(* PLC project PLCopen TC2 library, Higen Motion Controller 0.0 *)
(* stored: creationDateTime 2011-12-10T00:00:00, modificationDateTime 2011-12-10T00:00:00 *)

TYPE AXIS_REF : INT := -1;
END_TYPE

TYPE MC_BUFFER_MODE : (mcAborting, mcBuffered, mcBlendingLow, mcBlendingPrevious, mcBlendingNext, mcBlendingHigh) := mcAborting;
END_TYPE

TYPE MC_HOMING_PROCEDURES : (mcHomeDirect, mcHomeLimitSwitchPositive, mcHomeLimitSwitchNegative, mcHomeAbsoluteSwitchPositive, mcHomeAbsoluteSwitchNegative, mcHomeReferencePulsePositive, mcHomeReferencePulseNegative, mcHomeAbsolute) := mcHomeDirect;
END_TYPE

TYPE MC_DIRECTION : (mcAbsolutePosition, mcPositiveDirection, mcShortestWay, mcNegativeDirection, mcCurrentDirection) := mcAbsolutePosition;
END_TYPE

TYPE MC_TP_REF : INT := -1;
END_TYPE

TYPE MC_TV_REF : INT := -1;
END_TYPE

TYPE MC_TA_REF : INT := -1;
END_TYPE

TYPE MC_EXECUTION_MODE : (mcImmediately, mcQueued) := mcImmediately;
END_TYPE

TYPE MC_SOURCE : (mcActualValue, mcSetValue) := mcActualValue;
END_TYPE

TYPE MC_CAMSWITCH_REF : INT := -1;
END_TYPE

TYPE MC_OUTPUT_REF : INT := -1;
END_TYPE

TYPE MC_TRACK_REF : INT := -1;
END_TYPE

TYPE MC_TRIGGER_REF : INT := -1;
END_TYPE

TYPE MC_CAM_REF : INT := -1;
END_TYPE

TYPE MC_CAM_ID : INT := -1;
END_TYPE

TYPE MC_START_MODE : INT := -1;
END_TYPE

TYPE MC_SYNC_MODE : INT := -1;
END_TYPE

TYPE MC_COMBINE_MODE : (mcAddAxes, mcSubAxes) := mcAddAxes;
END_TYPE

TYPE MC_REAL_ARRAY : ARRAY[1..6] OF LREAL;
END_TYPE

TYPE MC_INT_ARRAY : ARRAY[1..6] OF INT;
END_TYPE

(* This fonction blocks returns the axis torque limits *)
FUNCTION_BLOCK MC_GetTorqueLimit
  VAR_IN_OUT
    Axis : AXIS_REF;
  END_VAR
  VAR_INPUT
    Execute : BOOL;
  END_VAR
  VAR_OUTPUT
    Done : BOOL;
    Busy : BOOL;
    Error : BOOL;
    ErrorID : WORD;
  END_VAR
  VAR_OUTPUT
    TorqueLimitPos : UINT;
    TorqueLimitNeg : UINT;
  END_VAR
  VAR
    Execute0 : BOOL;
    Done0 : BOOL;
  END_VAR

    {{
    extern void __mcl_cmd_MC_GetTorqueLimit(MC_GETTORQUELIMIT*);
    __mcl_cmd_MC_GetTorqueLimit(data__);
    }}
    Execute0 := Execute;
    Done0 := Done;
END_FUNCTION_BLOCK

(* This fonction blocks defines the axis torque limits *)
FUNCTION_BLOCK MC_SetTorqueLimit
  VAR_IN_OUT
    Axis : AXIS_REF;
  END_VAR
  VAR_INPUT
    Execute : BOOL;
  END_VAR
  VAR_OUTPUT
    Done : BOOL;
    Busy : BOOL;
    Error : BOOL;
    ErrorID : WORD;
  END_VAR
  VAR_INPUT
    TorqueLimitPos : UINT;
    TorqueLimitNeg : UINT;
  END_VAR
  VAR
    Execute0 : BOOL;
    Done0 : BOOL;
  END_VAR

    {{
    extern void __mcl_cmd_MC_SetTorqueLimit(MC_SETTORQUELIMIT*);
    __mcl_cmd_MC_SetTorqueLimit(data__);
    }}
    Execute0 := Execute;
    Done0 := Done;
END_FUNCTION_BLOCK

(* This Function Block controls the power stage (On or Off). *)
FUNCTION_BLOCK MC_Power
  VAR_IN_OUT
    Axis : AXIS_REF;
  END_VAR
  VAR_INPUT
    Enable : BOOL;
    EnablePositive : BOOL;
    EnableNegative : BOOL;
  END_VAR
  VAR_OUTPUT
    Status : BOOL;
    Valid : BOOL;
    Error : BOOL;
    ErrorID : WORD;
  END_VAR

    {{
    extern void __mcl_cmd_MC_Power(MC_POWER*);
    __mcl_cmd_MC_Power(data__);
    }}
END_FUNCTION_BLOCK

(* This Function Block commands the axis to perform the «search home» sequence. The details of this sequence are manufacturer dependent and can be set by the axis’ parameters. The ‘Position’ input is used to set the absolute position when reference signal is detected. This Function Block completes at ‘Standstill’ if it was started in ‘Standstill’. *)
FUNCTION_BLOCK MC_Home
  VAR_IN_OUT
    Axis : AXIS_REF;
  END_VAR
  VAR_INPUT
    Execute : BOOL;
    Position : LREAL;
    HomingMode : MC_HOMING_PROCEDURES;
    BufferMode : MC_BUFFER_MODE;
  END_VAR
  VAR_OUTPUT
    Done : BOOL;
    Busy : BOOL;
    Active : BOOL;
    CommandAborted : BOOL;
    Error : BOOL;
    ErrorID : WORD;
  END_VAR
  VAR
    Execute0 : BOOL;
    Done0 : BOOL;
    Active0 : BOOL;
  END_VAR

    {{
    extern void __mcl_cmd_MC_Home(MC_HOME*);
    __mcl_cmd_MC_Home(data__);
    }}
    Execute0 := Execute;
    Done0 := Done;
END_FUNCTION_BLOCK

(* This Function Block commands a controlled motion stop and transfers the axis to the state ‘Stopping’. It aborts any ongoing Function Block execution. While the axis is in state ‘Stopping’, no other FB can perform any motion on the same axis. After the axis has reached ‘Velocity’ zero, the ‘Done’ output is set to TRUE immediately. The axis remains in the state ‘Stopping’ as long as ‘Execute’ is still TRUE or ‘Velocity’ zero is not yet reached. As soon as ‘Done’ is SET and ‘Execute’ is FALSE the axis goes to state ‘Standstill’. *)
FUNCTION_BLOCK MC_Stop
  VAR_IN_OUT
    Axis : AXIS_REF;
  END_VAR
  VAR_INPUT
    Execute : BOOL;
    Deceleration : LREAL;
    Jerk : LREAL;
  END_VAR
  VAR_OUTPUT
    Done : BOOL;
    Busy : BOOL;
    CommandAborted : BOOL;
    Error : BOOL;
    ErrorID : WORD;
  END_VAR
  VAR
    Execute0 : BOOL;
    Done0 : BOOL;
    Active0 : BOOL;
  END_VAR

    {{
    extern void __mcl_cmd_MC_Stop(MC_STOP*);
    __mcl_cmd_MC_Stop(data__);
    }}
    Execute0 := Execute;
    Done0 := Done;
END_FUNCTION_BLOCK

(* This Function Block commands a controlled motion stop. The axis is moved to the state ‘DiscreteMotion’, until the velocity is zero. With the ‘Done’ output set, the state is transferred to ‘Standstill’. *)
FUNCTION_BLOCK MC_Halt
  VAR_IN_OUT
    Axis : AXIS_REF;
  END_VAR
  VAR_INPUT
    Execute : BOOL;
    Deceleration : LREAL;
    Jerk : LREAL;
    BufferMode : MC_BUFFER_MODE;
  END_VAR
  VAR_OUTPUT
    Done : BOOL;
    Busy : BOOL;
    Active : BOOL;
    CommandAborted : BOOL;
    Error : BOOL;
    ErrorID : WORD;
  END_VAR
  VAR
    Execute0 : BOOL;
    Done0 : BOOL;
    Active0 : BOOL;
  END_VAR

    {{
    extern void __mcl_cmd_MC_Halt(MC_HALT*);
    __mcl_cmd_MC_Halt(data__);
    }}
    Execute0 := Execute;
    Done0 := Done;
END_FUNCTION_BLOCK

(* This Function Block commands a controlled motion to a specified absolute position. *)
FUNCTION_BLOCK MC_MoveAbsolute
  VAR_IN_OUT
    Axis : AXIS_REF;
  END_VAR
  VAR_INPUT
    Execute : BOOL;
    ContinuousUpdate : BOOL;
    Position : LREAL;
    Velocity : LREAL;
    Acceleration : LREAL;
    Deceleration : LREAL;
    Jerk : LREAL;
    Direction : MC_DIRECTION;
    BufferMode : MC_BUFFER_MODE;
  END_VAR
  VAR_OUTPUT
    Done : BOOL;
    Busy : BOOL;
    Active : BOOL;
    CommandAborted : BOOL;
    Error : BOOL;
    ErrorID : WORD;
  END_VAR
  VAR
    Execute0 : BOOL;
    Done0 : BOOL;
    Active0 : BOOL;
  END_VAR

    {{
    extern void __mcl_cmd_MC_MoveAbsolute(MC_MOVEABSOLUTE*);
    __mcl_cmd_MC_MoveAbsolute(data__);
    }}
    Execute0 := Execute;
    Done0 := Done;
END_FUNCTION_BLOCK

(* This Function Block commands a controlled motion of a specified distance relative to the set position at the time of the execution. *)
FUNCTION_BLOCK MC_MoveRelative
  VAR_IN_OUT
    Axis : AXIS_REF;
  END_VAR
  VAR_INPUT
    Execute : BOOL;
    ContinuousUpdate : BOOL;
    Distance : LREAL;
    Velocity : LREAL;
    Acceleration : LREAL;
    Deceleration : LREAL;
    Jerk : LREAL;
    BufferMode : MC_BUFFER_MODE;
  END_VAR
  VAR_OUTPUT
    Done : BOOL;
    Busy : BOOL;
    Active : BOOL;
    CommandAborted : BOOL;
    Error : BOOL;
    ErrorID : WORD;
  END_VAR
  VAR
    Execute0 : BOOL;
    Done0 : BOOL;
    Active0 : BOOL;
  END_VAR

    {{
    extern void __mcl_cmd_MC_MoveRelative(MC_MOVERELATIVE*);
    __mcl_cmd_MC_MoveRelative(data__);
    }}
    Execute0 := Execute;
    Done0 := Done;
END_FUNCTION_BLOCK

(* This Function Block commands a controlled motion of a specified relative distance additional to the most recent commanded position in the axis state ‘DiscreteMotion’. The most recent commanded position may be the result of a previous MC_MoveAdditive motion which was aborted. If the FB is activated in the axis state ‘ContinuousMotion’, the specified relative distance is added to the set position at the time of the execution. *)
FUNCTION_BLOCK MC_MoveAdditive
  VAR_IN_OUT
    Axis : AXIS_REF;
  END_VAR
  VAR_INPUT
    Execute : BOOL;
    ContinuousUpdate : BOOL;
    Distance : LREAL;
    Velocity : LREAL;
    Acceleration : LREAL;
    Deceleration : LREAL;
    Jerk : LREAL;
    BufferMode : MC_BUFFER_MODE;
  END_VAR
  VAR_OUTPUT
    Done : BOOL;
    Busy : BOOL;
    Active : BOOL;
    CommandAborted : BOOL;
    Error : BOOL;
    ErrorID : WORD;
  END_VAR
  VAR
    Execute0 : BOOL;
    Done0 : BOOL;
    Active0 : BOOL;
  END_VAR

    {{
    extern void __mcl_cmd_MC_MoveAdditive(MC_MOVEADDITIVE*);
    __mcl_cmd_MC_MoveAdditive(data__);
    }}
    Execute0 := Execute;
    Done0 := Done;
END_FUNCTION_BLOCK

(* This Function Block commands a controlled motion of a specified relative distance additional to an existing motion. The existing Motion is not interrupted, but is superimposed by the additional motion. *)
FUNCTION_BLOCK MC_MoveSuperimposed
  VAR_IN_OUT
    Axis : AXIS_REF;
  END_VAR
  VAR_INPUT
    Execute : BOOL;
    ContinuousUpdate : BOOL;
    Distance : LREAL;
    VelocityDiff : LREAL;
    Acceleration : LREAL;
    Deceleration : LREAL;
    Jerk : LREAL;
  END_VAR
  VAR_OUTPUT
    Done : BOOL;
    Busy : BOOL;
    CommandAborted : BOOL;
    Error : BOOL;
    ErrorID : WORD;
    CoveredDistance : LREAL;
  END_VAR
  VAR
    Execute0 : BOOL;
    Done0 : BOOL;
    Active0 : BOOL;
  END_VAR

    {{
    extern void __mcl_cmd_MC_MoveSuperimposed(MC_MOVESUPERIMPOSED*);
    __mcl_cmd_MC_MoveSuperimposed(data__);
    }}
    Execute0 := Execute;
    Done0 := Done;
END_FUNCTION_BLOCK

(* This Function Block commands a halt to all superimposed motions of the axis. The underlying motion is not interrupted. *)
FUNCTION_BLOCK MC_HaltSuperimposed
  VAR_IN_OUT
    Axis : AXIS_REF;
  END_VAR
  VAR_INPUT
    Execute : BOOL;
    Deceleration : LREAL;
    Jerk : LREAL;
  END_VAR
  VAR_OUTPUT
    Done : BOOL;
    Busy : BOOL;
    CommandAborted : BOOL;
    Error : BOOL;
    ErrorID : WORD;
  END_VAR
  VAR
    Execute0 : BOOL;
    Done0 : BOOL;
    Active0 : BOOL;
  END_VAR

    {{
    extern void __mcl_cmd_MC_HaltSuperimposed(MC_HALTSUPERIMPOSED*);
    __mcl_cmd_MC_HaltSuperimposed(data__);
    }}
    Execute0 := Execute;
    Done0 := Done;
END_FUNCTION_BLOCK

(* This Function Block commands a never ending controlled motion at a specified velocity. *)
FUNCTION_BLOCK MC_MoveVelocity
  VAR_IN_OUT
    Axis : AXIS_REF;
  END_VAR
  VAR_INPUT
    Execute : BOOL;
    ContinuousUpdate : BOOL;
    Velocity : LREAL;
    Acceleration : LREAL;
    Deceleration : LREAL;
    Jerk : LREAL;
    Direction : MC_DIRECTION;
    BufferMode : MC_BUFFER_MODE;
  END_VAR
  VAR_OUTPUT
    InVelocity : BOOL;
    Busy : BOOL;
    Active : BOOL;
    CommandAborted : BOOL;
    Error : BOOL;
    ErrorID : WORD;
  END_VAR
  VAR
    Execute0 : BOOL;
    InVelocity0 : BOOL;
    Active0 : BOOL;
  END_VAR

    {{
    extern void __mcl_cmd_MC_MoveVelocity(MC_MOVEVELOCITY*);
    __mcl_cmd_MC_MoveVelocity(data__);
    }}
    Execute0 := Execute;
    InVelocity0 := InVelocity;
END_FUNCTION_BLOCK

(* This Function Block commands a controlled motion to a specified absolute position ending with the specified velocity. *)
FUNCTION_BLOCK MC_MoveContinuousAbsolute
  VAR_IN_OUT
    Axis : AXIS_REF;
  END_VAR
  VAR_INPUT
    Execute : BOOL;
    ContinuousUpdate : BOOL;
    Position : LREAL;
    EndVelocity : LREAL;
    Velocity : LREAL;
    Acceleration : LREAL;
    Deceleration : LREAL;
    Jerk : LREAL;
    Direction : MC_DIRECTION;
    BufferMode : MC_BUFFER_MODE;
  END_VAR
  VAR_OUTPUT
    InEndVelocity : BOOL;
    Busy : BOOL;
    Active : BOOL;
    CommandAborted : BOOL;
    Error : BOOL;
    ErrorID : WORD;
  END_VAR
  VAR
    Execute0 : BOOL;
    InEndVelocity0 : BOOL;
    Active0 : BOOL;
  END_VAR

    {{
    extern void __mcl_cmd_MC_MoveContinuousAbsolute(MC_MOVECONTINUOUSABSOLUTE*);
    __mcl_cmd_MC_MoveContinuousAbsolute(data__);
    }}
    Execute0 := Execute;
    InEndVelocity0 := InEndVelocity;
END_FUNCTION_BLOCK

(* This Function Block commands a controlled motion of a specified relative distance ending with the specified velocity. *)
FUNCTION_BLOCK MC_MoveContinuousRelative
  VAR_IN_OUT
    Axis : AXIS_REF;
  END_VAR
  VAR_INPUT
    Execute : BOOL;
    ContinuousUpdate : BOOL;
    Distance : LREAL;
    EndVelocity : LREAL;
    Velocity : LREAL;
    Acceleration : LREAL;
    Deceleration : LREAL;
    Jerk : LREAL;
    BufferMode : MC_BUFFER_MODE;
  END_VAR
  VAR_OUTPUT
    InEndVelocity : BOOL;
    Busy : BOOL;
    Active : BOOL;
    CommandAborted : BOOL;
    Error : BOOL;
    ErrorID : WORD;
  END_VAR
  VAR
    Execute0 : BOOL;
    InEndVelocity0 : BOOL;
    Active0 : BOOL;
  END_VAR

    {{
    extern void __mcl_cmd_MC_MoveContinuousRelative(MC_MOVECONTINUOUSRELATIVE*);
    __mcl_cmd_MC_MoveContinuousRelative(data__);
    }}
    Execute0 := Execute;
    InEndVelocity0 := InEndVelocity;
END_FUNCTION_BLOCK

(* This Function Block continuously exerts a torque or force of the specified magnitude. This magnitude is approached using a defined ramp (‘TorqueRamp’), and the Function Block sets the ‘InTorque’ output if the commanded torque level is reached. This function block is applicable for force and torque. When there is no external load, force is applicable. Positive torque is in the positive direction of velocity. *)
FUNCTION_BLOCK MC_TorqueControl
  VAR_IN_OUT
    Axis : AXIS_REF;
  END_VAR
  VAR_INPUT
    Execute : BOOL;
    ContinuousUpdate : BOOL;
    Torque : LREAL;
    TorqueRamp : LREAL;
    Velocity : LREAL;
    Acceleration : LREAL;
    Deceleration : LREAL;
    Jerk : LREAL;
    Direction : MC_DIRECTION;
    BufferMode : MC_BUFFER_MODE;
  END_VAR
  VAR_OUTPUT
    InTorque : BOOL;
    Busy : BOOL;
    Active : BOOL;
    CommandAborted : BOOL;
    Error : BOOL;
    ErrorID : WORD;
  END_VAR
  VAR
    Execute0 : BOOL;
    InTorque0 : BOOL;
    Active0 : BOOL;
  END_VAR

    {{
    extern void __mcl_cmd_MC_TorqueControl(MC_TORQUECONTROL*);
    __mcl_cmd_MC_TorqueControl(data__);
    }}
    Execute0 := Execute;
    InTorque0 := InTorque;
END_FUNCTION_BLOCK

(* This Function Block commands a time-position locked motion profile *)
FUNCTION_BLOCK MC_PositionProfile
  VAR_IN_OUT
    Axis : AXIS_REF;
    TimePosition : MC_TP_REF;
  END_VAR
  VAR_INPUT
    Execute : BOOL;
    ContinuousUpdate : BOOL;
    TimeScale : LREAL := 1.0;
    PositionScale : LREAL := 1.0;
    Offset : LREAL;
    BufferMode : MC_BUFFER_MODE;
  END_VAR
  VAR_OUTPUT
    Done : BOOL;
    Busy : BOOL;
    Active : BOOL;
    CommandAborted : BOOL;
    Error : BOOL;
    ErrorID : WORD;
  END_VAR
  VAR
    Execute0 : BOOL;
    Done0 : BOOL;
    Active0 : BOOL;
  END_VAR

    {{
    extern void __mcl_cmd_MC_PositionProfile(MC_POSITIONPROFILE*);
    __mcl_cmd_MC_PositionProfile(data__);
    }}
    Execute0 := Execute;
    Done0 := Done;
END_FUNCTION_BLOCK

(* This Function Block commands a time-velocity locked motion profile. The velocity in the final element in the profile should be maintained. The state remains ‘ContinuousMotion’. *)
FUNCTION_BLOCK MC_VelocityProfile
  VAR_IN_OUT
    Axis : AXIS_REF;
    TimeVelocity : MC_TV_REF;
  END_VAR
  VAR_INPUT
    Execute : BOOL;
    ContinuousUpdate : BOOL;
    TimeScale : LREAL := 1.0;
    VelocityScale : LREAL := 1.0;
    Offset : LREAL;
    BufferMode : MC_BUFFER_MODE;
  END_VAR
  VAR_OUTPUT
    ProfileCompleted : BOOL;
    Busy : BOOL;
    Active : BOOL;
    CommandAborted : BOOL;
    Error : BOOL;
    ErrorID : WORD;
  END_VAR
  VAR
    Execute0 : BOOL;
    ProfileCompleted0 : BOOL;
    Active0 : BOOL;
  END_VAR

    {{
    extern void __mcl_cmd_MC_VelocityProfile(MC_VELOCITYPROFILE*);
    __mcl_cmd_MC_VelocityProfile(data__);
    }}
    Execute0 := Execute;
    ProfileCompleted0 := ProfileCompleted;
END_FUNCTION_BLOCK

(* This Function Block commands a time-acceleration locked motion profile. After finalizing the acceleration profile, the acceleration goes to 0 (and typically the final velocity is maintained). It stays in the state ‘ContinuousMotion’. *)
FUNCTION_BLOCK MC_AccelerationProfile
  VAR_IN_OUT
    Axis : AXIS_REF;
    TimeAcceleration : MC_TA_REF;
  END_VAR
  VAR_INPUT
    Execute : BOOL;
    ContinuousUpdate : BOOL;
    TimeScale : LREAL := 1.0;
    AccelerationScale : LREAL := 1.0;
    Offset : LREAL;
    BufferMode : MC_BUFFER_MODE;
  END_VAR
  VAR_OUTPUT
    ProfileCompleted : BOOL;
    Busy : BOOL;
    Active : BOOL;
    CommandAborted : BOOL;
    Error : BOOL;
    ErrorID : WORD;
  END_VAR
  VAR
    Execute0 : BOOL;
    ProfileCompleted0 : BOOL;
    Active0 : BOOL;
  END_VAR

    {{
    extern void __mcl_cmd_MC_AccelerationProfile(MC_ACCELERATIONPROFILE*);
    __mcl_cmd_MC_AccelerationProfile(data__);
    }}
    Execute0 := Execute;
    ProfileCompleted0 := ProfileCompleted;
END_FUNCTION_BLOCK

(* This Function Block shifts the coordinate system of an axis by manipulating both the set-point position as well as the actual position of an axis with the same value without any movement caused. (Re-calibration with same following error). This can be used for instance for a reference situation. This Function Block can also be used during motion without changing the commanded position, which is now positioned in the shifted coordinate system. *)
FUNCTION_BLOCK MC_SetPosition
  VAR_IN_OUT
    Axis : AXIS_REF;
  END_VAR
  VAR_INPUT
    Execute : BOOL;
    Position : LREAL;
    Relative : BOOL;
    ExecutionMode : MC_EXECUTION_MODE;
  END_VAR
  VAR_OUTPUT
    Done : BOOL;
    Busy : BOOL;
    Error : BOOL;
    ErrorID : WORD;
  END_VAR
  VAR
    Execute0 : BOOL;
    Done0 : BOOL;
  END_VAR

    {{
    extern void __mcl_cmd_MC_SetPosition(MC_SETPOSITION*);
    __mcl_cmd_MC_SetPosition(data__);
    }}
    Execute0 := Execute;
    Done0 := Done;
END_FUNCTION_BLOCK

(* This Function Block sets the values of override for the whole axis, and all functions that are working on that axis. The override parameters contribute as a factor to the calculation of the commanded velocity, acceleration and jerk of the motion. *)
FUNCTION_BLOCK MC_SetOverride
  VAR_IN_OUT
    Axis : AXIS_REF;
  END_VAR
  VAR_INPUT
    Enable : BOOL;
    VelFactor : LREAL := 1.0;
    AccFactor : LREAL := 1.0;
    JerkFactor : LREAL := 1.0;
  END_VAR
  VAR_OUTPUT
    Enabled : BOOL;
    Busy : BOOL;
    Error : BOOL;
    ErrorID : WORD;
  END_VAR
  VAR
    Enable0 : BOOL;
  END_VAR

    {{
    extern void __mcl_cmd_MC_SetOverride(MC_SETOVERRIDE*);
    __mcl_cmd_MC_SetOverride(data__);
    }}
    Enable0 := Enable;
END_FUNCTION_BLOCK

(* This Function Block returns the value of a vendor specific parameter. The returned Value has to be converted to Real if necessary. If not possible, the vendor has to supply a vendor specific FB to read the parameter. *)
FUNCTION_BLOCK MC_ReadParameter
  VAR_IN_OUT
    Axis : AXIS_REF;
  END_VAR
  VAR_INPUT
    Enable : BOOL;
    ParameterNumber : INT;
  END_VAR
  VAR_OUTPUT
    Valid : BOOL;
    Busy : BOOL;
    Error : BOOL;
    ErrorID : WORD;
    Value : LREAL;
  END_VAR
  VAR
    Enable0 : BOOL;
  END_VAR

    {{
    extern void __mcl_cmd_MC_ReadParameter(MC_READPARAMETER*);
    __mcl_cmd_MC_ReadParameter(data__);
    }}
    Enable0 := Enable;
END_FUNCTION_BLOCK

(* This Function Block returns the value of a vendor specific parameter with datatype BOOL. *)
FUNCTION_BLOCK MC_ReadBoolParameter
  VAR_IN_OUT
    Axis : AXIS_REF;
  END_VAR
  VAR_INPUT
    Enable : BOOL;
    ParameterNumber : INT;
  END_VAR
  VAR_OUTPUT
    Valid : BOOL;
    Busy : BOOL;
    Error : BOOL;
    ErrorID : WORD;
    Value : BOOL;
  END_VAR
  VAR
    Enable0 : BOOL;
  END_VAR

    {{
    extern void __mcl_cmd_MC_ReadBoolParameter(MC_READBOOLPARAMETER*);
    __mcl_cmd_MC_ReadBoolParameter(data__);
    }}
    Enable0 := Enable;
END_FUNCTION_BLOCK

(* This Function Block modifies the value of a vendor specific parameter. *)
FUNCTION_BLOCK MC_WriteParameter
  VAR_IN_OUT
    Axis : AXIS_REF;
  END_VAR
  VAR_INPUT
    Execute : BOOL;
    ParameterNumber : INT;
    Value : LREAL;
    ExecutionMode : MC_EXECUTION_MODE;
  END_VAR
  VAR_OUTPUT
    Done : BOOL;
    Busy : BOOL;
    Error : BOOL;
    ErrorID : WORD;
  END_VAR
  VAR
    Execute0 : BOOL;
    Done0 : BOOL;
  END_VAR

    {{
    extern void __mcl_cmd_MC_WriteParameter(MC_WRITEPARAMETER*);
    __mcl_cmd_MC_WriteParameter(data__);
    }}
    Execute0 := Execute;
    Done0 := Done;
END_FUNCTION_BLOCK

(* This Function Block modifies the value of a vendor specific parameter of type BOOL. *)
FUNCTION_BLOCK MC_WriteBoolParameter
  VAR_IN_OUT
    Axis : AXIS_REF;
  END_VAR
  VAR_INPUT
    Execute : BOOL;
    ParameterNumber : INT;
    Value : BOOL;
    ExecutionMode : MC_EXECUTION_MODE;
  END_VAR
  VAR_OUTPUT
    Done : BOOL;
    Busy : BOOL;
    Error : BOOL;
    ErrorID : WORD;
  END_VAR
  VAR
    Execute0 : BOOL;
    Done0 : BOOL;
  END_VAR

    {{
    extern void __mcl_cmd_MC_WriteBoolParameter(MC_WRITEBOOLPARAMETER*);
    __mcl_cmd_MC_WriteBoolParameter(data__);
    }}
    Execute0 := Execute;
    Done0 := Done;
END_FUNCTION_BLOCK

(* This Function Block gives access to the value of the input, referenced by the datatype AXIS_REF. It provides the value of the referenced input (BOOL) *)
FUNCTION_BLOCK MC_ReadDigitalInput
  VAR_IN_OUT
    Input : AXIS_REF;
  END_VAR
  VAR_INPUT
    Enable : BOOL;
    InputNumber : INT;
  END_VAR
  VAR_OUTPUT
    Valid : BOOL;
    Busy : BOOL;
    Error : BOOL;
    ErrorID : WORD;
    Value : BOOL;
  END_VAR
  VAR
    Enable0 : BOOL;
  END_VAR

    {{
    extern void __mcl_cmd_MC_ReadDigitalInput(MC_READDIGITALINPUT*);
    __mcl_cmd_MC_ReadDigitalInput(data__);
    }}
    Enable0 := Enable;
END_FUNCTION_BLOCK

(* This Function Block provides access to the value of a digital output, referenced by the datatype AXIS_REF. It provides the value of the referenced output (BOOL). *)
FUNCTION_BLOCK MC_ReadDigitalOutput
  VAR_IN_OUT
    Output : AXIS_REF;
  END_VAR
  VAR_INPUT
    Enable : BOOL;
    OutputNumber : INT;
  END_VAR
  VAR_OUTPUT
    Valid : BOOL;
    Busy : BOOL;
    Error : BOOL;
    ErrorID : WORD;
    Value : BOOL;
  END_VAR
  VAR
    Enable0 : BOOL;
  END_VAR

    {{
    extern void __mcl_cmd_MC_ReadDigitalOutput(MC_READDIGITALOUTPUT*);
    __mcl_cmd_MC_ReadDigitalOutput(data__);
    }}
    Enable0 := Enable;
END_FUNCTION_BLOCK

(* This Function Block writes a value to the output referenced by the argument ‘Output’ once (with rising edge of Execute). *)
FUNCTION_BLOCK MC_WriteDigitalOutput
  VAR_IN_OUT
    Output : AXIS_REF;
  END_VAR
  VAR_INPUT
    Execute : BOOL;
    OutputNumber : INT;
    Value : BOOL;
    ExecutionMode : MC_EXECUTION_MODE;
  END_VAR
  VAR_OUTPUT
    Done : BOOL;
    Busy : BOOL;
    Error : BOOL;
    ErrorID : WORD;
  END_VAR
  VAR
    Execute0 : BOOL;
    Done0 : BOOL;
  END_VAR

    {{
    extern void __mcl_cmd_MC_WriteDigitalOutput(MC_WRITEDIGITALOUTPUT*);
    __mcl_cmd_MC_WriteDigitalOutput(data__);
    }}
    Execute0 := Execute;
    Done0 := Done;
END_FUNCTION_BLOCK

(* This Function Block returns the actual position. *)
FUNCTION_BLOCK MC_ReadActualPosition
  VAR_IN_OUT
    Axis : AXIS_REF;
  END_VAR
  VAR_INPUT
    Enable : BOOL;
  END_VAR
  VAR_OUTPUT
    Valid : BOOL;
    Busy : BOOL;
    Error : BOOL;
    ErrorID : WORD;
    Position : LREAL;
  END_VAR
  VAR
    Enable0 : BOOL;
  END_VAR

    {{
    extern void __mcl_cmd_MC_ReadActualPosition(MC_READACTUALPOSITION*);
    __mcl_cmd_MC_ReadActualPosition(data__);
    }}
    Enable0 := Enable;
END_FUNCTION_BLOCK

(* This Function Block returns the value of the actual velocity as long as ‘Enable’ is set. ‘Valid’ is true when the dataoutput ‘Velocity’ is valid. If ‘Enable’ is Reset, the data loses its validity, and all outputs are reset, no matter if new data is available. *)
FUNCTION_BLOCK MC_ReadActualVelocity
  VAR_IN_OUT
    Axis : AXIS_REF;
  END_VAR
  VAR_INPUT
    Enable : BOOL;
  END_VAR
  VAR_OUTPUT
    Valid : BOOL;
    Busy : BOOL;
    Error : BOOL;
    ErrorID : WORD;
    Velocity : LREAL;
  END_VAR
  VAR
    Enable0 : BOOL;
  END_VAR

    {{
    extern void __mcl_cmd_MC_ReadActualVelocity(MC_READACTUALVELOCITY*);
    __mcl_cmd_MC_ReadActualVelocity(data__);
    }}
    Enable0 := Enable;
END_FUNCTION_BLOCK

(* This Function Block returns the value of the actual torque or force as long as ‘Enable’ is set. ‘Valid’ is true when the data-output ‘Torque’ is valid. If ‘Enable’ is Reset, the data loses its validity, and ‘Valid’ is also reset, no matter if new data is available. *)
FUNCTION_BLOCK MC_ReadActualTorque
  VAR_IN_OUT
    Axis : AXIS_REF;
  END_VAR
  VAR_INPUT
    Enable : BOOL;
  END_VAR
  VAR_OUTPUT
    Valid : BOOL;
    Busy : BOOL;
    Error : BOOL;
    ErrorID : WORD;
    Torque : LREAL;
  END_VAR
  VAR
    Enable0 : BOOL;
  END_VAR

    {{
    extern void __mcl_cmd_MC_ReadActualTorque(MC_READACTUALTORQUE*);
    __mcl_cmd_MC_ReadActualTorque(data__);
    }}
    Enable0 := Enable;
END_FUNCTION_BLOCK

(* This Function Block returns in detail the status of the state diagram of the selected axis. *)
FUNCTION_BLOCK MC_ReadStatus
  VAR_IN_OUT
    Axis : AXIS_REF;
  END_VAR
  VAR_INPUT
    Enable : BOOL;
  END_VAR
  VAR_OUTPUT
    Valid : BOOL;
    Busy : BOOL;
    Error : BOOL;
    ErrorID : WORD;
    ErrorStop : BOOL;
    Disabled : BOOL;
    Stopping : BOOL;
    Homing : BOOL;
    Standstill : BOOL;
    DiscreteMotion : BOOL;
    ContinuousMotion : BOOL;
    SynchronizedMotion : BOOL;
  END_VAR
  VAR
    Enable0 : BOOL;
  END_VAR

    {{
    extern void __mcl_cmd_MC_ReadStatus(MC_READSTATUS*);
    __mcl_cmd_MC_ReadStatus(data__);
    }}
    Enable0 := Enable;
END_FUNCTION_BLOCK

(* This Function Block returns in detail the status of the axis with respect to the motion currently in progress. *)
FUNCTION_BLOCK MC_ReadMotionState
  VAR_IN_OUT
    Axis : AXIS_REF;
  END_VAR
  VAR_INPUT
    Enable : BOOL;
    Source : MC_SOURCE;
  END_VAR
  VAR_OUTPUT
    Valid : BOOL;
    Busy : BOOL;
    Error : BOOL;
    ErrorID : WORD;
    ConstantVelocity : BOOL;
    Accelerating : BOOL;
    Decelerating : BOOL;
    DirectionPositive : BOOL;
    DirectionNegative : BOOL;
  END_VAR
  VAR
    Enable0 : BOOL;
  END_VAR

    {{
    extern void __mcl_cmd_MC_ReadMotionState(MC_READMOTIONSTATE*);
    __mcl_cmd_MC_ReadMotionState(data__);
    }}
    Enable0 := Enable;
END_FUNCTION_BLOCK

(* This Function Block reads information concerning an axis, like modes, inputs directly related to the axis, and certain status information. *)
FUNCTION_BLOCK MC_ReadAxisInfo
  VAR_IN_OUT
    Axis : AXIS_REF;
  END_VAR
  VAR_INPUT
    Enable : BOOL;
  END_VAR
  VAR_OUTPUT
    Valid : BOOL;
    Busy : BOOL;
    Error : BOOL;
    ErrorID : WORD;
    HomeAbsSwitch : BOOL;
    LimitSwitchPos : BOOL;
    LimitSwitchNeg : BOOL;
    Simulation : BOOL;
    CommunicationReady : BOOL;
    ReadyForPowerOn : BOOL;
    PowerOn : BOOL;
    IsHomed : BOOL;
    AxisWarning : BOOL;
  END_VAR
  VAR
    Enable0 : BOOL;
  END_VAR

    {{
    extern void __mcl_cmd_MC_ReadAxisInfo(MC_READAXISINFO*);
    __mcl_cmd_MC_ReadAxisInfo(data__);
    }}
    Enable0 := Enable;
END_FUNCTION_BLOCK

(* This Function Block presents general axis errors not relating to the Function Blocks. (for instance axis errors, drive errors, communication errors) *)
FUNCTION_BLOCK MC_ReadAxisError
  VAR_IN_OUT
    Axis : AXIS_REF;
  END_VAR
  VAR_INPUT
    Enable : BOOL;
  END_VAR
  VAR_OUTPUT
    Valid : BOOL;
    Busy : BOOL;
    Error : BOOL;
    ErrorID : WORD;
    AxisErrorID : WORD;
  END_VAR
  VAR
    Enable0 : BOOL;
  END_VAR

    {{
    extern void __mcl_cmd_MC_ReadAxisError(MC_READAXISERROR*);
    __mcl_cmd_MC_ReadAxisError(data__);
    }}
    Enable0 := Enable;
END_FUNCTION_BLOCK

(* This Function Block makes the transition from the state ‘ErrorStop’ to ‘Standstill’ or ‘Disabled’ by resetting all internal axis-related errors – it does not affect the output of the FB instances. *)
FUNCTION_BLOCK MC_Reset
  VAR_IN_OUT
    Axis : AXIS_REF;
  END_VAR
  VAR_INPUT
    Execute : BOOL;
  END_VAR
  VAR_OUTPUT
    Done : BOOL;
    Busy : BOOL;
    Error : BOOL;
    ErrorID : WORD;
  END_VAR
  VAR
    Execute0 : BOOL;
    Done0 : BOOL;
  END_VAR

    {{
    extern void __mcl_cmd_MC_Reset(MC_RESET*);
    __mcl_cmd_MC_Reset(data__);
    }}
    Execute0 := Execute;
    Done0 := Done;
END_FUNCTION_BLOCK

(* This Function Block is the analogy to switches on a motor shaft: it commands a group of discrete output bits to switch in analogy to a set of mechanical cam controlled switches connected to an axis. Forward and backward movements are allowed. *)
FUNCTION_BLOCK MC_DigitalCamSwitch
  VAR_IN_OUT
    Axis : AXIS_REF;
    Switches : MC_CAMSWITCH_REF;
    Outputs : MC_OUTPUT_REF;
    TrackOptions : MC_TRACK_REF;
  END_VAR
  VAR_INPUT
    Enable : BOOL;
    EnableMask : DWORD;
    ValueSource : MC_SOURCE;
  END_VAR
  VAR_OUTPUT
    InOperation : BOOL;
    Busy : BOOL;
    Error : BOOL;
    ErrorID : WORD;
  END_VAR
  VAR
    Enable0 : BOOL;
    InOperation0 : BOOL;
  END_VAR

    {{
    extern void __mcl_cmd_MC_DigitalCamSwitch(MC_DIGITALCAMSWITCH*);
    __mcl_cmd_MC_DigitalCamSwitch(data__);
    }}
    Enable0 := Enable;
    InOperation0 := InOperation;
END_FUNCTION_BLOCK

(* This Function Block is used to record an axis position at a trigger event *)
FUNCTION_BLOCK MC_TouchProbe
  VAR_IN_OUT
    Axis : AXIS_REF;
    TriggerInput : MC_TRIGGER_REF;
  END_VAR
  VAR_INPUT
    Execute : BOOL;
    WindowOnly : BOOL;
    FirstPosition : LREAL;
    LastPosition : LREAL;
  END_VAR
  VAR_OUTPUT
    Done : BOOL;
    Busy : BOOL;
    CommandAborted : BOOL;
    Error : BOOL;
    ErrorID : WORD;
    RecordedPosition : LREAL;
  END_VAR
  VAR
    Execute0 : BOOL;
    Done0 : BOOL;
    Active0 : BOOL;
  END_VAR

    {{
    extern void __mcl_cmd_MC_TouchProbe(MC_TOUCHPROBE*);
    __mcl_cmd_MC_TouchProbe(data__);
    }}
    Execute0 := Execute;
    Done0 := Done;
END_FUNCTION_BLOCK

(* This Function Block is used to abort function blocks which are connected to trigger events (e.g. MC_TouchProbe) *)
FUNCTION_BLOCK MC_AbortTrigger
  VAR_IN_OUT
    Axis : AXIS_REF;
    TriggerInput : MC_TRIGGER_REF;
  END_VAR
  VAR_INPUT
    Execute : BOOL;
  END_VAR
  VAR_OUTPUT
    Done : BOOL;
    Busy : BOOL;
    Error : BOOL;
    ErrorID : WORD;
  END_VAR
  VAR
    Execute0 : BOOL;
    Done0 : BOOL;
  END_VAR

    {{
    extern void __mcl_cmd_MC_AbortTrigger(MC_ABORTTRIGGER*);
    __mcl_cmd_MC_AbortTrigger(data__);
    }}
    Execute0 := Execute;
    Done0 := Done;
END_FUNCTION_BLOCK

(* This Function Block selects the CAM tables by setting the connections to the relevant tables *)
FUNCTION_BLOCK MC_CamTableSelect
  VAR_IN_OUT
    Master : AXIS_REF;
    Slave : AXIS_REF;
    CamTable : MC_CAM_REF;
  END_VAR
  VAR_INPUT
    Execute : BOOL;
    Periodic : BOOL;
    MasterAbsolute : BOOL;
    SlaveAbsolute : BOOL;
    ExecutionMode : MC_EXECUTION_MODE;
  END_VAR
  VAR_OUTPUT
    Done : BOOL;
    Busy : BOOL;
    Error : BOOL;
    ErrorID : WORD;
    CamTableID : MC_CAM_ID;
  END_VAR
  VAR
    Execute0 : BOOL;
    Done0 : BOOL;
    RefInit : BOOL;
    CamTableIDRef : MC_CAM_ID;
  END_VAR

    IF NOT(RefInit) THEN
      {{
          extern int __MK_Alloc_MC_CAM_ID();
          int res=__MK_Alloc_MC_CAM_ID();
          SetFbVar(CAMTABLEID,res);
          SetFbVar(CAMTABLEIDREF,res);
      }}
      RefInit := TRUE;
    END_IF;
    {{
    extern void __mcl_cmd_MC_CamTableSelect(MC_CAMTABLESELECT*);
    __mcl_cmd_MC_CamTableSelect(data__);
    }}
    Execute0 := Execute;
    Done0 := Done;
END_FUNCTION_BLOCK

(* This Function Block engages the CAM *)
FUNCTION_BLOCK MC_CamIn
  VAR_IN_OUT
    Master : AXIS_REF;
    Slave : AXIS_REF;
  END_VAR
  VAR_INPUT
    Execute : BOOL;
    ContinuousUpdate : BOOL;
    MasterOffset : LREAL;
    SlaveOffset : LREAL;
    MasterScaling : LREAL := 1.0;
    SlaveScaling : LREAL := 1.0;
    MasterStartDistance : LREAL;
    MasterSyncPosition : LREAL;
    StartMode : MC_START_MODE;
    MasterValueSource : MC_SOURCE;
    CamTableID : MC_CAM_ID;
    BufferMode : MC_BUFFER_MODE;
  END_VAR
  VAR_OUTPUT
    InSync : BOOL;
    Busy : BOOL;
    Active : BOOL;
    CommandAborted : BOOL;
    Error : BOOL;
    ErrorID : WORD;
    EndOfProfile : BOOL;
  END_VAR
  VAR
    Execute0 : BOOL;
    InSync0 : BOOL;
    Active0 : BOOL;
  END_VAR

    {{
    extern void __mcl_cmd_MC_CamIn(MC_CAMIN*);
    __mcl_cmd_MC_CamIn(data__);
    }}
    Execute0 := Execute;
    InSync0 := InSync;
END_FUNCTION_BLOCK

(* This Function Block disengages the Slave axis from the Master axis immediately *)
FUNCTION_BLOCK MC_CamOut
  VAR_IN_OUT
    Slave : AXIS_REF;
  END_VAR
  VAR_INPUT
    Execute : BOOL;
  END_VAR
  VAR_OUTPUT
    Done : BOOL;
    Busy : BOOL;
    Error : BOOL;
    ErrorID : WORD;
  END_VAR
  VAR
    Execute0 : BOOL;
    Done0 : BOOL;
  END_VAR

    {{
    extern void __mcl_cmd_MC_CamOut(MC_CAMOUT*);
    __mcl_cmd_MC_CamOut(data__);
    }}
    Execute0 := Execute;
    Done0 := Done;
END_FUNCTION_BLOCK

(* This Function Block commands a ratio between the VELOCITY of the slave and master axis. *)
FUNCTION_BLOCK MC_GearIn
  VAR_IN_OUT
    Master : AXIS_REF;
    Slave : AXIS_REF;
  END_VAR
  VAR_INPUT
    Execute : BOOL;
    ContinuousUpdate : BOOL;
    RatioNumerator : INT := 1;
    RatioDenominator : UINT := 1;
    MasterValueSource : MC_SOURCE;
    Acceleration : LREAL;
    Deceleration : LREAL;
    Jerk : LREAL;
    BufferMode : MC_BUFFER_MODE;
  END_VAR
  VAR_OUTPUT
    InGear : BOOL;
    Busy : BOOL;
    Active : BOOL;
    CommandAborted : BOOL;
    Error : BOOL;
    ErrorID : WORD;
  END_VAR
  VAR
    Execute0 : BOOL;
    InGear0 : BOOL;
    Active0 : BOOL;
  END_VAR

    {{
    extern void __mcl_cmd_MC_GearIn(MC_GEARIN*);
    __mcl_cmd_MC_GearIn(data__);
    }}
    Execute0 := Execute;
    InGear0 := InGear;
END_FUNCTION_BLOCK

(* This Function Block disengages the Slave axis from the Master axis *)
FUNCTION_BLOCK MC_GearOut
  VAR_IN_OUT
    Slave : AXIS_REF;
  END_VAR
  VAR_INPUT
    Execute : BOOL;
  END_VAR
  VAR_OUTPUT
    Done : BOOL;
    Busy : BOOL;
    Error : BOOL;
    ErrorID : WORD;
  END_VAR
  VAR
    Execute0 : BOOL;
    Done0 : BOOL;
  END_VAR

    {{
    extern void __mcl_cmd_MC_GearOut(MC_GEAROUT*);
    __mcl_cmd_MC_GearOut(data__);
    }}
    Execute0 := Execute;
    Done0 := Done;
END_FUNCTION_BLOCK

(* This Function Block commands a gear ratio between the position of the slave and master axes from the synchronization point onwards. *)
FUNCTION_BLOCK MC_GearInPos
  VAR_IN_OUT
    Master : AXIS_REF;
    Slave : AXIS_REF;
  END_VAR
  VAR_INPUT
    Execute : BOOL;
    RatioNumerator : INT := 1;
    RatioDenominator : UINT := 1;
    MasterValueSource : MC_SOURCE;
    MasterSyncPosition : LREAL;
    SlaveSyncPosition : LREAL;
    SyncMode : MC_SYNC_MODE;
    MasterStartDistance : LREAL;
    Velocity : LREAL;
    Acceleration : LREAL;
    Deceleration : LREAL;
    Jerk : LREAL;
    BufferMode : MC_BUFFER_MODE;
  END_VAR
  VAR_OUTPUT
    StartSync : BOOL;
    InSync : BOOL;
    Busy : BOOL;
    Active : BOOL;
    CommandAborted : BOOL;
    Error : BOOL;
    ErrorID : WORD;
  END_VAR
  VAR
    Execute0 : BOOL;
    InSync0 : BOOL;
    Active0 : BOOL;
  END_VAR

    {{
    extern void __mcl_cmd_MC_GearInPos(MC_GEARINPOS*);
    __mcl_cmd_MC_GearInPos(data__);
    }}
    Execute0 := Execute;
    InSync0 := InSync;
END_FUNCTION_BLOCK

(* This Function Block creates an absolute phase shift in the master position of a slave axis. The master position is shifted in relation to the real physical position. This is analogous to opening a coupling on the master shaft for a moment, and is used to delay or advance an axis to its master. The phase shift is seen from the slave. The master does not know that there is a phase shift experienced by the slave (MasterPos as seen from the SlaveAxis = PhysicalMasterPos + PhaseShiftValueSlaveAxis, the phase shift value has the character of a position offset) The phase shift remains until another ‘Phasing’ command changes it again. *)
FUNCTION_BLOCK MC_PhasingAbsolute
  VAR_IN_OUT
    Master : AXIS_REF;
    Slave : AXIS_REF;
  END_VAR
  VAR_INPUT
    Execute : BOOL;
    PhaseShift : LREAL;
    Velocity : LREAL;
    Acceleration : LREAL;
    Deceleration : LREAL;
    Jerk : LREAL;
    BufferMode : MC_BUFFER_MODE;
  END_VAR
  VAR_OUTPUT
    Done : BOOL;
    Busy : BOOL;
    Active : BOOL;
    CommandAborted : BOOL;
    Error : BOOL;
    ErrorID : WORD;
    AbsolutePhaseShift : LREAL;
  END_VAR
  VAR
    Execute0 : BOOL;
    Done0 : BOOL;
    Active0 : BOOL;
  END_VAR

    {{
    extern void __mcl_cmd_MC_PhasingAbsolute(MC_PHASINGABSOLUTE*);
    __mcl_cmd_MC_PhasingAbsolute(data__);
    }}
    Execute0 := Execute;
    Done0 := Done;
END_FUNCTION_BLOCK

(* This Function Block creates a phase shift in the master position of a slave axis relative to the existing phase shift. The master position is shifted in relation to the real physical position. This is analogous to opening a coupling on the master shaft for a moment, and is used to delay or advance an axis to its master. The phase shift is seen from the slave. The master does not know that there is a phase shift experienced by the slave. (MasterPos as seen from SlaveAxis = PhysicalMasterPos + PhaseShiftValueSlaveAxis, the phase shift value has the character of a position offset) The phase shift remains until another ‘Phasing’ command changes it again. Relative phase shifts are added to each other for the applicable phase shift *)
FUNCTION_BLOCK MC_PhasingRelative
  VAR_IN_OUT
    Master : AXIS_REF;
    Slave : AXIS_REF;
  END_VAR
  VAR_INPUT
    Execute : BOOL;
    PhaseShift : LREAL;
    Velocity : LREAL;
    Acceleration : LREAL;
    Deceleration : LREAL;
    Jerk : LREAL;
    BufferMode : MC_BUFFER_MODE;
  END_VAR
  VAR_OUTPUT
    Done : BOOL;
    Busy : BOOL;
    Active : BOOL;
    CommandAborted : BOOL;
    Error : BOOL;
    ErrorID : WORD;
    CoveredPhaseShift : LREAL;
  END_VAR
  VAR
    Execute0 : BOOL;
    Done0 : BOOL;
    Active0 : BOOL;
  END_VAR

    {{
    extern void __mcl_cmd_MC_PhasingRelative(MC_PHASINGRELATIVE*);
    __mcl_cmd_MC_PhasingRelative(data__);
    }}
    Execute0 := Execute;
    Done0 := Done;
END_FUNCTION_BLOCK

(* This Function Block combines the motion of 2 axes into a third axis with selectable combination method. Basically it is a calculation of a new position setpoint based on the 2 position setpoints of the input axes. This FB is reflected in the state diagram like a synchronized motion type. As application example one can work with a separate profile synchronized to an object on a moving belt, or a rotating knife with flexible covered distance to be cut. *)
FUNCTION_BLOCK MC_CombineAxes
  VAR_IN_OUT
    Master1 : AXIS_REF;
    Master2 : AXIS_REF;
    Slave : AXIS_REF;
  END_VAR
  VAR_INPUT
    Execute : BOOL;
    ContinuousUpdate : BOOL;
    CombineMode : MC_COMBINE_MODE;
    GearRatioNumeratorM1 : INT := 1;
    GearRatioDenominatorM1 : INT := 1;
    GearRatioNumeratorM2 : INT := 1;
    GearRatioDenominatorM2 : INT := 1;
    MasterValueSourceM1 : MC_SOURCE;
    MasterValueSourceM2 : MC_SOURCE;
    BufferMode : MC_BUFFER_MODE;
  END_VAR
  VAR_OUTPUT
    InSync : BOOL;
    Busy : BOOL;
    Active : BOOL;
    CommandAborted : BOOL;
    Error : BOOL;
    ErrorID : WORD;
  END_VAR
  VAR
    Execute0 : BOOL;
    InSync0 : BOOL;
    Active0 : BOOL;
  END_VAR

    {{
    extern void __mcl_cmd_MC_CombineAxes(MC_COMBINEAXES*);
    __mcl_cmd_MC_CombineAxes(data__);
    }}
    Execute0 := Execute;
    InSync0 := InSync;
END_FUNCTION_BLOCK

(* This allocates a simulation Axis, for testing. One axis per instanciated FB. *)
FUNCTION_BLOCK MC_Sim
  VAR_INPUT
    MaxVel : LREAL := 1.0;
    MaxAcc : LREAL := 1.0;
    MaxDec : LREAL := 1.0;
  END_VAR
  VAR_OUTPUT
    Axis : AXIS_REF;
  END_VAR
  VAR
    SimParam : MC_WriteBoolParameter;
    VelParam : MC_WriteParameter;
    AccParam : MC_WriteParameter;
    DecParam : MC_WriteParameter;
    Done : BOOL;
  END_VAR

IF NOT Done THEN
  {{
    extern int __MK_Alloc_AXIS_REF(); 
    int res=__MK_Alloc_AXIS_REF();
    __SET_VAR(data__->,AXIS,res);
  }}
  SimParam(Axis := Axis,
           Execute := BOOL#TRUE,
           ParameterNumber := 1000, 
           Value := BOOL#TRUE);
  VelParam(Axis := Axis,
           Execute := BOOL#TRUE,
           ParameterNumber := 9,
           Value := MaxVel);
  AccParam(Axis := Axis, 
           Execute := BOOL#TRUE,
           ParameterNumber := 13,
           Value := MaxAcc);
  DecParam(Axis := Axis,
           Execute := BOOL#TRUE,
           ParameterNumber := 15,
           Value := MaxDec);
  Done := TRUE;
END_IF;
END_FUNCTION_BLOCK

(* Create MC_TRIGGER_REF type, with given parameters. PositiveEdge and NegativeEdged default to TRUE. *)
FUNCTION_BLOCK MC_CreateTrigger
  VAR_INPUT
    PositiveEdge : BOOL := TRUE;
    NegativeEdge : BOOL := TRUE;
  END_VAR
  VAR_OUTPUT
    TriggerInput : MC_TRIGGER_REF;
  END_VAR
  VAR
    Done : BOOL;
  END_VAR

IF NOT Done THEN
  {{
  extern int __MK_Alloc_MC_TRIGGER_REF();
  extern char* __MK_GetPublic_MC_TRIGGER_REF(int);
  int res=__MK_Alloc_MC_TRIGGER_REF(); 
  if(res>=0) 
      *__MK_GetPublic_MC_TRIGGER_REF(res)=
         (GetFbVar(POSITIVEEDGE) ? 0x01 : 0)
        |(GetFbVar(NEGATIVEEDGE) ? 0x02 : 0);
  SetFbVar(TRIGGERINPUT,res); 
  }}
  Done := TRUE;
END_IF;
END_FUNCTION_BLOCK

(* This allocates an output object. One output per instanciated FB. *)
FUNCTION_BLOCK MC_CreateOutput
  VAR_OUTPUT
    Output : MC_OUTPUT_REF;
  END_VAR
  VAR
    Done : BOOL;
  END_VAR

IF NOT Done THEN
  {{
      extern int __MK_Alloc_MC_OUTPUT_REF();
      int res=__MK_Alloc_MC_OUTPUT_REF();
      SetFbVar(OUTPUT,res);
  }}
  Done := TRUE;
END_IF;
END_FUNCTION_BLOCK

(* This generate an array of 6 INT from inputs. *)
FUNCTION_BLOCK MC_ToIntArray
  VAR_OUTPUT
    IntArray : MC_INT_ARRAY;
  END_VAR
  VAR_INPUT
    X : INT;
    Y : INT;
    Z : INT;
    U : INT;
    V : INT;
    W : INT;
  END_VAR

IntArray[1]:=X;
IntArray[2]:=Y;
IntArray[3]:=Z;
IntArray[4]:=U;
IntArray[5]:=V;
IntArray[6]:=W;
END_FUNCTION_BLOCK

(* This returns bits contained in MC_OUTPUT_REF. *)
FUNCTION_BLOCK MC_ReadOutputBits
  VAR_OUTPUT
    Bits : DWORD;
  END_VAR
  VAR_INPUT
    Output : MC_OUTPUT_REF;
  END_VAR

{{
extern uint32_t* __MK_GetPublic_MC_OUTPUT_REF(int);
SetFbVar(BITS, *__MK_GetPublic_MC_OUTPUT_REF(GetFbVar(OUTPUT)));
}}
END_FUNCTION_BLOCK

(* This returns bits contained in MC_OUTPUT_REF. *)
FUNCTION_BLOCK MC_ReadOutputBit
  VAR_OUTPUT
    Bit : BOOL;
  END_VAR
  VAR_INPUT
    Output : MC_OUTPUT_REF;
    OutputNumber : INT;
  END_VAR

{{
extern uint32_t* __MK_GetPublic_MC_OUTPUT_REF(int);
SetFbVar(BIT, (*__MK_GetPublic_MC_OUTPUT_REF(GetFbVar(OUTPUT)) >> 
GetFbVar(OUTPUTNUMBER)) & 1);
}}
END_FUNCTION_BLOCK

(* Load a CSV file, and present it as variable of type MC_TP_REF. *)
FUNCTION_BLOCK MC_TP_REF_FROM_CSV
  VAR_INPUT
    FileName : STRING;
  END_VAR
  VAR_OUTPUT
    Active : BOOL;
    Valid : BOOL;
    TimeProfile : MC_TP_REF;
  END_VAR
  VAR
    py1 : python_eval;
  END_VAR

IF NOT Active THEN
  {{
    extern int __MK_Alloc_MC_TP_REF();
    int res=__MK_Alloc_MC_TP_REF();
    SetFbVar(TIMEPROFILE,res);
  }}
  Active := TRUE;
END_IF;
py1(TRIG := TRUE, CODE := CONCAT('MK_Load_MC_TP_REF_CSV(', INT_TO_STRING(TimeProfile),',"', FileName, '")'));
IF AND(py1.ACK, EQ(py1.RESULT, 'True')) THEN
  {{
    extern uint8_t __MK_CheckPublic_MC_TP_REF(int);
    if (__MK_CheckPublic_MC_TP_REF(GetFbVar(TIMEPROFILE))){
        SetFbVar(VALID,TRUE);
    }
  }}
END_IF;
END_FUNCTION_BLOCK

(* Load a CSV file, and present it as variable of type MC_TV_REF. *)
FUNCTION_BLOCK MC_TV_REF_FROM_CSV
  VAR_INPUT
    FileName : STRING;
  END_VAR
  VAR_OUTPUT
    Active : BOOL;
    Valid : BOOL;
    TimeProfile : MC_TV_REF;
  END_VAR
  VAR
    py1 : python_eval;
  END_VAR

IF NOT Active THEN
  {{
    extern int __MK_Alloc_MC_TV_REF();
    int res=__MK_Alloc_MC_TV_REF();
    SetFbVar(TIMEPROFILE,res);
  }}
  Active := TRUE;
END_IF;
py1(TRIG := TRUE, CODE := CONCAT('MK_Load_MC_TV_REF_CSV(', INT_TO_STRING(TimeProfile),',"', FileName, '")'));
IF AND(py1.ACK, EQ(py1.RESULT, 'True')) THEN
  {{
    extern uint8_t __MK_CheckPublic_MC_TV_REF(int);
    if (__MK_CheckPublic_MC_TV_REF(GetFbVar(TIMEPROFILE))){
        SetFbVar(VALID,TRUE);
    }
  }}
END_IF;
END_FUNCTION_BLOCK

(* Load a CSV file, and present it as variable of type MC_TA_REF. *)
FUNCTION_BLOCK MC_TA_REF_FROM_CSV
  VAR_INPUT
    FileName : STRING;
  END_VAR
  VAR_OUTPUT
    Active : BOOL;
    Valid : BOOL;
    TimeProfile : MC_TA_REF;
  END_VAR
  VAR
    py1 : python_eval;
  END_VAR

IF NOT Active THEN
  {{
    extern int __MK_Alloc_MC_TA_REF();
    int res=__MK_Alloc_MC_TA_REF();
    SetFbVar(TIMEPROFILE,res);
  }}
  Active := TRUE;
END_IF;
py1(TRIG := TRUE, CODE := CONCAT('MK_Load_MC_TA_REF_CSV(', INT_TO_STRING(TimeProfile),',"', FileName, '")'));
IF AND(py1.ACK, EQ(py1.RESULT, 'True')) THEN
  {{
    extern uint8_t __MK_CheckPublic_MC_TA_REF(int);
    if (__MK_CheckPublic_MC_TA_REF(GetFbVar(TIMEPROFILE))){
        SetFbVar(VALID,TRUE);
    }
  }}
END_IF;
END_FUNCTION_BLOCK

(* Load a CSV file, and present it as variable of type MC_CAMSWITCH_REF. *)
FUNCTION_BLOCK MC_CAMSWITCH_REF_FROM_CSV
  VAR_INPUT
    FileName : STRING;
  END_VAR
  VAR_OUTPUT
    Active : BOOL;
    Valid : BOOL;
    CamSwitchList : MC_CAMSWITCH_REF;
  END_VAR
  VAR
    py1 : python_eval;
  END_VAR

IF NOT Active THEN
  {{
    extern int __MK_Alloc_MC_CAMSWITCH_REF();
    int res=__MK_Alloc_MC_CAMSWITCH_REF();
    SetFbVar(CAMSWITCHLIST,res);
  }}
  Active := TRUE;
END_IF;
py1(TRIG := TRUE, CODE := CONCAT('MK_Load_MC_CAMSWITCH_REF_CSV(', INT_TO_STRING(CamSwitchList),',"', FileName, '")'));
IF AND(py1.ACK, EQ(py1.RESULT, 'True')) THEN
  {{
    extern uint8_t __MK_CheckPublic_MC_CAMSWITCH_REF(int);
    if (__MK_CheckPublic_MC_CAMSWITCH_REF(GetFbVar(CAMSWITCHLIST))){
        SetFbVar(VALID,TRUE);
    }
  }}
END_IF;
END_FUNCTION_BLOCK

(* Load a CSV file, and present it as variable of type MC_CAM_REF. *)
FUNCTION_BLOCK MC_CAM_REF_FROM_CSV
  VAR_INPUT
    FileName : STRING;
  END_VAR
  VAR_OUTPUT
    Active : BOOL;
    Valid : BOOL;
    CamTable : MC_CAM_REF;
  END_VAR
  VAR
    py1 : python_eval;
  END_VAR

IF NOT Active THEN
  {{
    extern int __MK_Alloc_MC_CAM_REF();
    int res=__MK_Alloc_MC_CAM_REF();
    SetFbVar(CAMTABLE,res);
  }}
  Active := TRUE;
END_IF;
py1(TRIG := TRUE, CODE := CONCAT('MK_Load_MC_CAM_REF_CSV(', INT_TO_STRING(CamTable),',"', FileName, '")'));
IF AND(py1.ACK, EQ(py1.RESULT, 'True')) THEN
  {{
    extern uint8_t __MK_CheckPublic_MC_CAM_REF(int);
    if (__MK_CheckPublic_MC_CAM_REF(GetFbVar(CAMTABLE))){
        SetFbVar(VALID,TRUE);
    }
  }}
END_IF;
END_FUNCTION_BLOCK
